# EPICS autosave request: iocBoot/iocVindum/auto_settings.req
file "VindumController_settings.req" P=$(P)
file "VindumPumpN_settings.req",     P=$(P), PUMP=A:
file "VindumPumpN_settings.req",     P=$(P), PUMP=B:
